% RSLogix 500 project RAILWAY GATE_BAK012.RSS, saved by version 8.30.00.16 %
PROJECT "UNTITLED"    % processor: MicroLogix 1000 %

PROGRAM FILES
  LAD 2 "MAIN_PROG"  11 rungs
  LAD 3 "USER_FAULT"  1 rungs
  LAD 4 "HSC_INT"  1 rungs
  LAD 5 "STI_INT"  1 rungs
  LAD 6, 7, 8, 9, 10, 11, 12, 13, 14, 15, 16: only END

DATA FILES
  O0 OUTPUT  1 elements
  I1 INPUT  2 elements
  S2 STATUS  33 elements
  B3 BINARY  32 elements
  T4 TIMER  40 elements
  C5 COUNTER  32 elements
  R6 CONTROL  16 elements
  N7 INTEGER  105 elements

LADDER 2 "MAIN_PROG"
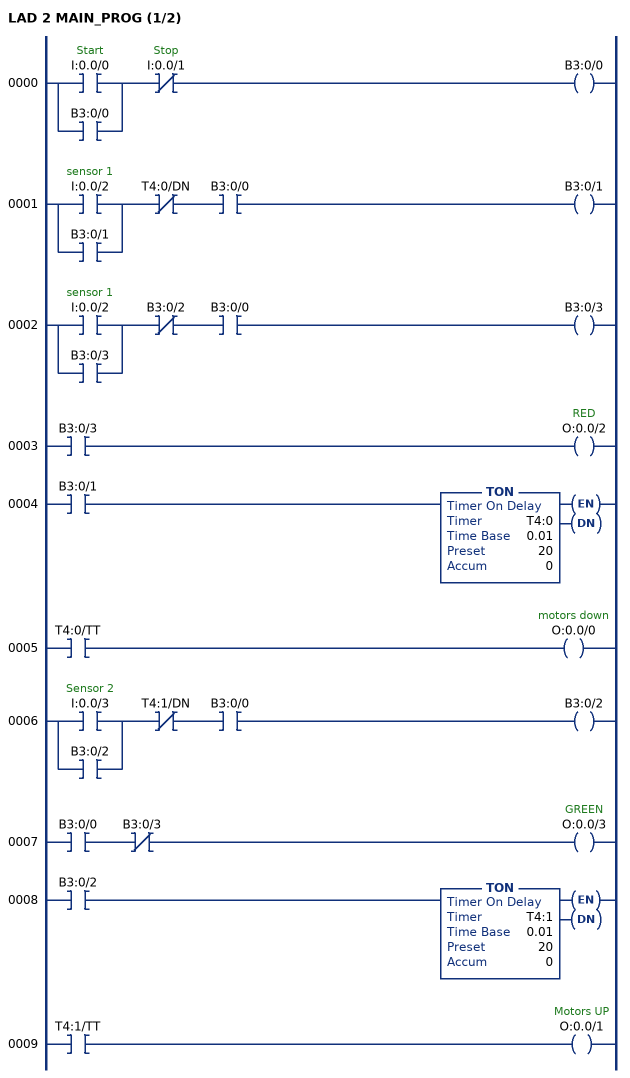
% Rung: 0 %
SOR BST XIC I:0.0/0 NXB XIC B3:0/0 BND XIO I:0.0/1 OTE B3:0/0 EOR
%   I:0.0/0  "Start" %
%   I:0.0/1  "Stop" %
% Rung: 1 %
SOR BST XIC I:0.0/2 NXB XIC B3:0/1 BND XIO T4:0/DN XIC B3:0/0 OTE B3:0/1 EOR
%   I:0.0/2  "sensor 1" %
% Rung: 2 %
SOR BST XIC I:0.0/2 NXB XIC B3:0/3 BND XIO B3:0/2 XIC B3:0/0 OTE B3:0/3 EOR
%   I:0.0/2  "sensor 1" %
% Rung: 3 %
SOR XIC B3:0/3 OTE O:0.0/2 EOR
%   O:0.0/2  "RED" %
% Rung: 4 %
SOR XIC B3:0/1 TON T4:0 0.01 20 0 EOR
% Rung: 5 %
SOR XIC T4:0/TT OTE O:0.0/0 EOR
%   O:0.0/0  "motors down" %
% Rung: 6 %
SOR BST XIC I:0.0/3 NXB XIC B3:0/2 BND XIO T4:1/DN XIC B3:0/0 OTE B3:0/2 EOR
%   I:0.0/3  "Sensor 2" %
% Rung: 7 %
SOR XIC B3:0/0 XIO B3:0/3 OTE O:0.0/3 EOR
%   O:0.0/3  "GREEN" %
% Rung: 8 %
SOR XIC B3:0/2 TON T4:1 0.01 20 0 EOR
% Rung: 9 %
SOR XIC T4:1/TT OTE O:0.0/1 EOR
%   O:0.0/1  "Motors UP" %

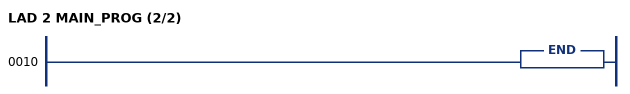
% Rung: 10 %
SOR END EOR

DATA TABLE (non-zero values as saved)
DATA B3
% B3:0 % 0X0001 0X0000 0X0000 0X0000 0X0000 0X0000 0X0000 0X0000 0X0000 0X0000
DATA T4
% .PRE .ACC %
% T4:0 % 20 0
% T4:1 % 20 0
